// TIA Portal V18 export
FUNCTION_BLOCK "MOTOR"   // FB17, LAD
{ S7_Optimized_Access := 'TRUE' }
VERSION : 0.1
// stored: AutoNumber true, IsIECCheckEnabled false, IsRetainMemResEnabled false, MemoryReserve 100, SetENOAutomatically false, UDAEnableTagReadback false
   VAR_INPUT
      "auto/manual" : Bool;
      auto_on : Bool;
      manual_on : Bool;
      run_fb : Bool;
      stop_fb : Bool;
      reset : Bool;
      intl : Bool;
      Mon_En : Bool;
      mon_sp : Time;
      trip : Bool;
   END_VAR
   VAR_OUTPUT
      running : Bool;
      fault : Bool;
      status : Int;
      Off_relay : Bool;
   END_VAR
   VAR
      on_fault : Bool;
      off_fault : Bool;
      IEC_Timer_0_Instance : TON_TIME;
      IEC_Timer_0_Instance_1 { S7_SetPoint := 'True'} : TON_TIME;
      mon { S7_SetPoint := 'True'} : Int;
      pulse : Bool;
      pulse1 : Bool;
      mon1 : Int;
      IEC_Timer_0_Instance_2 : TON_TIME;
      off_pls : Bool;
      Off_relay_bit : Bool;
      timer1 { S7_SetPoint := 'True'} : TON_TIME;
   END_VAR
   VAR_TEMP   // added for the SCL form of the ladder/FBD networks
      _w1 : Bool;
      _w2 : Bool;
   END_VAR
BEGIN

REGION Network 1
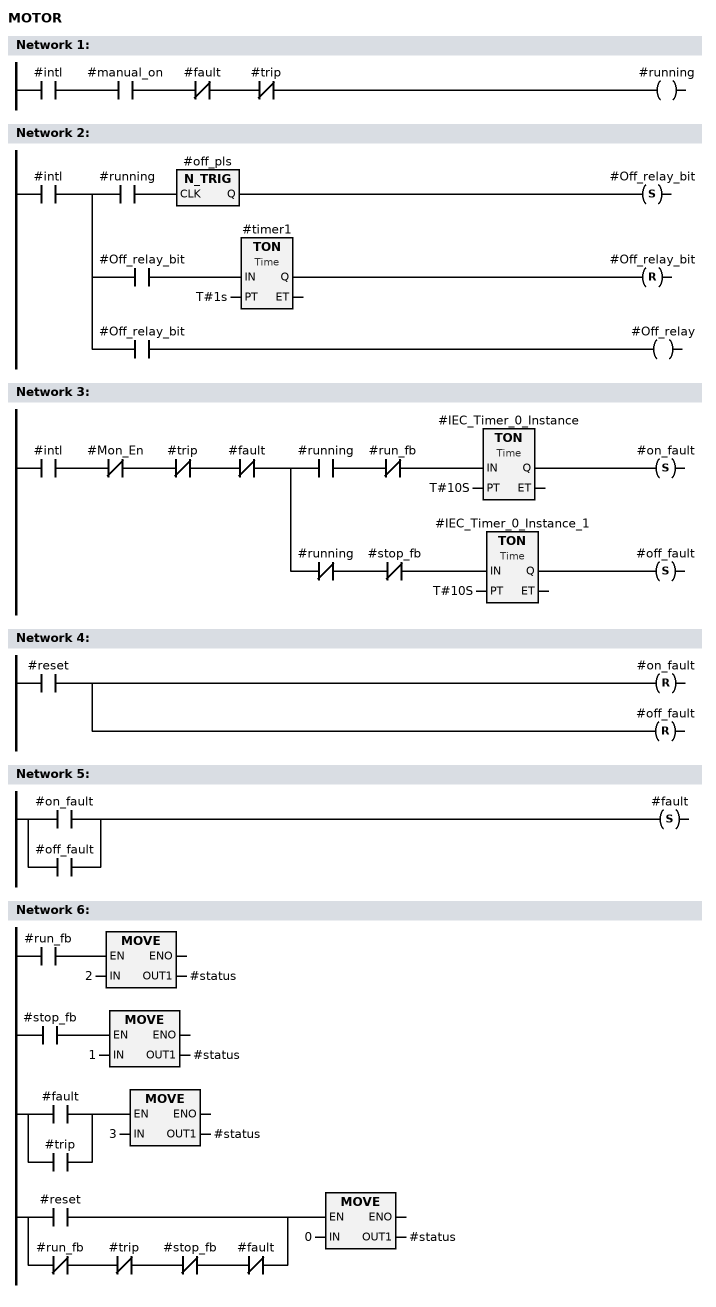
   RUNG wire#powerrail
      Contact( #intl )
      Contact( #manual_on )
      I_Contact( #fault )
      I_Contact( #trip )
      Coil( #running )
   END_RUNG
   // the same network as SCL:
   #running := #intl AND #manual_on AND NOT #fault AND NOT #trip;
END_REGION

REGION Network 2
   RUNG wire#powerrail
      Contact( #intl )
      wire#w1
      Contact( #running )
      N_Trig( #off_pls )
      S_Coil( #Off_relay_bit )
   END_RUNG
   RUNG wire#w1
      Contact( #Off_relay_bit )
      { S7_Templates := "time_type := Time" } #timer1.TON(pt := T#1s, et =>)
      R_Coil( #Off_relay_bit )
   END_RUNG
   RUNG wire#w1
      Contact( #Off_relay_bit )
      Coil( #Off_relay )
   END_RUNG
   // the same network as SCL:
   #_w1 := #intl AND #running;
   #_w2 := NOT #_w1 AND #off_pls;   // falling edge
   #off_pls := #_w1;
   IF #_w2 THEN #Off_relay_bit := TRUE; END_IF;
   #timer1(IN := #intl AND #Off_relay_bit, PT := T#1s);   // TON
   IF #timer1.Q THEN #Off_relay_bit := FALSE; END_IF;
   #Off_relay := #intl AND #Off_relay_bit;
END_REGION

REGION Network 3
   RUNG wire#powerrail
      Contact( #intl )
      I_Contact( #Mon_En )
      I_Contact( #trip )
      I_Contact( #fault )
      wire#w1
      Contact( #running )
      I_Contact( #run_fb )
      { S7_Templates := "time_type := Time" } #IEC_Timer_0_Instance.TON(pt := T#10S, et =>)
      S_Coil( #on_fault )
   END_RUNG
   RUNG wire#w1
      I_Contact( #running )
      I_Contact( #stop_fb )
      { S7_Templates := "time_type := Time" } #IEC_Timer_0_Instance_1.TON(pt := T#10S, et =>)
      S_Coil( #off_fault )
   END_RUNG
   // the same network as SCL:
   #_w1 := #intl AND NOT #Mon_En AND NOT #trip AND NOT #fault;
   #IEC_Timer_0_Instance(IN := #_w1 AND #running AND NOT #run_fb, PT := T#10S);   // TON
   IF #IEC_Timer_0_Instance.Q THEN #on_fault := TRUE; END_IF;
   #IEC_Timer_0_Instance_1(IN := #_w1 AND NOT #running AND NOT #stop_fb, PT := T#10S);   // TON
   IF #IEC_Timer_0_Instance_1.Q THEN #off_fault := TRUE; END_IF;
END_REGION

REGION Network 4
   RUNG wire#powerrail
      Contact( #reset )
      wire#w1
      R_Coil( #on_fault )
   END_RUNG
   RUNG wire#w1
      R_Coil( #off_fault )
   END_RUNG
   // the same network as SCL:
   IF #reset THEN
       #on_fault := FALSE;
       #off_fault := FALSE;
   END_IF;
END_REGION

REGION Network 5
   RUNG wire#powerrail
      Contact( #on_fault )
      wire#w1
      S_Coil( #fault )
   END_RUNG
   RUNG wire#powerrail
      Contact( #off_fault )
   END_RUNG wire#w1
   // the same network as SCL:
   IF #on_fault OR #off_fault THEN #fault := TRUE; END_IF;
END_REGION

REGION Network 6
   RUNG wire#powerrail
      Contact( #run_fb )
      Move(in := 2, out1 => #status)
   END_RUNG
   RUNG wire#powerrail
      Contact( #stop_fb )
      Move(in := 1, out1 => #status)
   END_RUNG
   RUNG wire#powerrail
      Contact( #fault )
      wire#w1
      Move(in := 3, out1 => #status)
   END_RUNG
   RUNG wire#powerrail
      Contact( #trip )
   END_RUNG wire#w1
   RUNG wire#powerrail
      Contact( #reset )
      wire#w2
      Move(in := 0, out1 => #status)
   END_RUNG
   RUNG wire#powerrail
      I_Contact( #run_fb )
      I_Contact( #trip )
      I_Contact( #stop_fb )
      I_Contact( #fault )
   END_RUNG wire#w2
   // the same network as SCL:
   IF #run_fb THEN #status := 2; END_IF;
   IF #stop_fb THEN #status := 1; END_IF;
   IF #fault OR #trip THEN #status := 3; END_IF;
   IF #reset OR (NOT #run_fb AND NOT #trip AND NOT #stop_fb AND NOT #fault) THEN #status := 0; END_IF;
END_REGION
END_FUNCTION_BLOCK
